{attribute 'qualified_only'}
{attribute 'strict'}
{attribute 'to_string'}
TYPE e_db_steel_local :
(
	holdingEntranceRack := 1, // 吊掛入料區
	entranceRack := 2, // 入料區
	machine := 10, // 機台內
	holdingExitRack := 20, // 吊掛出料區
	exitRack := 21 // 出料區
);
END_TYPE
//  exitRack = '21 '

(* stored: Version 1.1.0.1, ProductVersion 3.1.4026.13
   EnumerationTextList e_db_steel_local: Id {e10f3d5d-10e4-469a-a72b-75d522f29ac0} *)
